TYPE UDT 1000
TITLE =PLC ==> 611U Process Data (POS Mode Control)
VERSION : 0.1


  STRUCT
   STW1 : STRUCT
    Bit_8 : BOOL ;	//Jog 1 On/Off
    Bit_9 : BOOL ;	//Jog 2 On/Off
    Bit_10 : BOOL ;	//Control Requested / No Control Requested
    Bit_11 : BOOL ;	//Start Referencing / Stop Referencing
    Bit_12 : BOOL ;	//Reserved
    Bit_13 : BOOL ;	//External Block Change
    Bit_14 : BOOL ;	//Reserved
    Bit_15 : BOOL ;	//Reserved
    Bit_0 : BOOL ;	//Enable / Off 1
    Bit_1 : BOOL ;	//Enable / Off 2
    Bit_2 : BOOL ;	//Enable / Off 3
    Bit_3 : BOOL ;	//Enable Inverter / Pulse Inhibit
    Bit_4 : BOOL ;	//Enable / Reject travel task
    Bit_5 : BOOL ;	//Enable / Immediatly stop
    Bit_6 : BOOL ;	//Activate Travel Block ( Edge )
    Bit_7 : BOOL ;	//Reset the Fault memory
   END_STRUCT ;
   SatzAnw : STRUCT
    BLKSEL : INT ;	//Block Selection 0 ~ 63
   END_STRUCT ;
   PosStw : STRUCT
    Bit_8 : BOOL ;	//Reserved
    Bit_9 : BOOL ;	//Reserved
    Bit_10 : BOOL ;	//Reserved
    Bit_11 : BOOL ;	//Reserved
    Bit_12 : BOOL ;	//Reserved
    Bit_13 : BOOL ;	//Reserved
    Bit_14 : BOOL ;	//Reserved
    Bit_15 : BOOL ;	//Reserved
    Bit_0 : BOOL ;	//Tracking Operation
    Bit_1 : BOOL ;	//Set Reference Point
    Bit_2 : BOOL ;	//Reference Cams
    Bit_3 : BOOL ;	//Acknowledgement, Function Bit
    Bit_4 : BOOL ;	//Reserved
    Bit_5 : BOOL ;	//Reserved
    Bit_6 : BOOL ;	//Reserved
    Bit_7 : BOOL ;	//Reserved
   END_STRUCT ;
   STW2 : STRUCT
    Bit_8 : BOOL ;	//Suppress Fault 608
    Bit_9 : BOOL ;	//Motor Data Change Over 1st input
    Bit_10 : BOOL ;	//Motor Data Change Over 2nd input
    Bit_11 : BOOL ;	//Motor Changed Over
    Bit_12 : BOOL ;	//Sign of Life Bit 0
    Bit_13 : BOOL ;	//Sign of Life Bit 1
    Bit_14 : BOOL ;	//Sign of Life Bit 2
    Bit_15 : BOOL ;	//Sign of Life Bit 3
    Bit_0 : BOOL ;	//Parameter Set Changeover Bit 0
    Bit_1 : BOOL ;	//Parameter Set Changeover Bit 1
    Bit_2 : BOOL ;	//Parameter Set Changeover Bit 2
    Bit_3 : BOOL ;	//First Speed Setpoint Filter off
    Bit_4 : BOOL ;	//Ramp up Time Zero
    Bit_5 : BOOL ;	//Reserved
    Bit_6 : BOOL ;	//Integrator inhibit, Speed Controller
    Bit_7 : BOOL ;	//Selection, Parking Axis
   END_STRUCT ;
   Over : STRUCT
    Override : INT ;	//Override Defined using P0833=>16384(dec) = 1%, 1638.4 = 0.1%
   END_STRUCT ;
   Temp1 : INT ;
   Temp2 : INT ;
   Temp3 : INT ;
   Temp4 : INT ;
   Temp5 : INT ;
  END_STRUCT ;
END_TYPE

TYPE UDT 2000
TITLE =POS Mode Control
VERSION : 0.1


  STRUCT
   ZSW1 : STRUCT
    Bit_8 : BOOL ;	//No Following error / Following error
    Bit_9 : BOOL ;	//Control requested / No Control Possible
    Bit_10 : BOOL ;	//Reference Point Reached / Outside ref.position
    Bit_11 : BOOL ;	//Reference Point Set / Reference Point Not Set
    Bit_12 : BOOL ;	//Setpoint Acknowledge (Edge)
    Bir_13 : BOOL ;	//Drive Stationary / Drive Active
    Bit_14 : BOOL ;	//Reserved
    Bit_15 : BOOL ;	//Reserved
    Bit_0 : BOOL ;	//Ready to Switch-on / Not ready to Switch-on
    Bit_1 : BOOL ;	//Ready or no Fault
    Bit_2 : BOOL ;	//Controller Enable Status
    Bit_3 : BOOL ;	//Fault Present / No Fault Present
    Bit_4 : BOOL ;	//No OFF2 Present / OFF2 Present
    Bit_5 : BOOL ;	//No OFF3 Present / OFF3 Present
    Bit_6 : BOOL ;	//Switch-on Inhibit / No Switch-on Inhibit
    Bit_7 : BOOL ;	//Alarm Present / No Alarm Present
   END_STRUCT ;
   AktSatz : STRUCT
    CURRBLK : INT ;	//Status Block Selection (0 ~ 63)
   END_STRUCT ;
   PosZsw : STRUCT
    Bit_8 : BOOL ;	//Cam Switching Signal 1
    Bit_9 : BOOL ;	//Cam Switching Signal 2
    Bit_10 : BOOL ;	//Direct Output 1 via the Traversing Block
    Bit_11 : BOOL ;	//Direct Output 2 via the Traversing Block
    Bit_12 : BOOL ;	//Reserved
    Bit_13 : BOOL ;	//Reserved
    Bit_14 : BOOL ;	//Reserved
    Bit_15 : BOOL ;	//Reserved
    Bit_0 : BOOL ;	//Tracking Mode Active
    Bit_1 : BOOL ;	//Velocity Limiting
    Bit_2 : BOOL ;	//Setpoint stationary
    Bit_3 : BOOL ;	//Function Bit
    Bit_4 : BOOL ;	//Axis Moves Forwards
    Bit_5 : BOOL ;	//Axis Moves Backwards
    Bit_6 : BOOL ;	//Minus Software Limit Switch Actuated
    Bit_7 : BOOL ;	//Plus Software Limit Switch Actuated
   END_STRUCT ;
   ZSW2 : STRUCT
    Bit_8 : BOOL ;	//Supress Fault 608 Active
    Bit_9 : BOOL ;	//Actual Motor 1st Signal
    Bit_10 : BOOL ;	//Actual Motor 2nd Signal
    Bit_11 : BOOL ;	//Reserved
    Bit_12 : BOOL ;	//Slave Sign of Life Bit 0
    Bit_13 : BOOL ;	//Slave Sign of Life Bit 1
    Bit_14 : BOOL ;	//Slave Sign of Life Bit 2
    Bit_15 : BOOL ;	//Slave Sign of Life Bit 3
    Bit_0 : BOOL ;	//Parameter Set Bit 0
    Bit_1 : BOOL ;	//Parameter Set Bit 1
    Bit_2 : BOOL ;	//Parameter Set Bit 2
    Bit_3 : BOOL ;	//First Speed Setpoint Filter Inactive
    Bit_4 : BOOL ;	//Ramp-Function gen Inactive
    Bit_5 : BOOL ;	//Open Holding Brake
    Bit_6 : BOOL ;	//Integrator Inhibit, Speed Controller
    Bit_7 : BOOL ;	//Parking Axis Selected
   END_STRUCT ;
   MessW : STRUCT
    Bit_8 : BOOL ;	//|nset| = |nact |
    Bit_9 : BOOL ;	//Reserved
    Bit_10 : BOOL ;	//Power Module Current Not Limited
    Bit_11 : BOOL ;	//Reserved
    Bit_12 : BOOL ;	//Reserved
    Bit_13 : BOOL ;	//Pulse Enabled
    Bit_14 : BOOL ;	//Reserved
    Bit_15 : BOOL ;	//Reserved
    Bit_0 : BOOL ;	//Ramp-up Completed
    Bit_1 : BOOL ;	//|M| < Mx
    Bit_2 : BOOL ;	//|nact| < nmin
    Bit_3 : BOOL ;	//|nact| < nx
    Bit_4 : BOOL ;	//DC Link Monitoring VDC link > Vx
    Bit_5 : BOOL ;	//Variable Message Function
    Bit_6 : BOOL ;	//Motor Overtemperature Pre-Alarm
    Bit_7 : BOOL ;	//Heatsink Temperature Pre-Alarm
   END_STRUCT ;
   XactP1 : WORD ;	//Position Actual Value (Pos Mode) Word1
   XactP2 : WORD ;	//Position Actual Value (Pos Mode) Word2
   Temp1 : INT ;
   Temp2 : INT ;
   Temp3 : INT ;
  END_STRUCT ;
END_TYPE

DATA_BLOCK DB 2
TITLE =
VERSION : 0.1


  STRUCT
   SEND1_DATA : STRUCT 	//Temporary placeholder variable
    SEND_DONE : BOOL ;
    SEND_ERROR : BOOL ;
    SEND_SCAN : BOOL ;
    SEND_ACT : BOOL ;
    SEND_SP1 : BOOL ;
    SEND_SP2 : BOOL ;
    SEND_SP3 : BOOL ;
    SEND_SP4 : BOOL ;
    SEND_STATUS : WORD ;
    SPARE2 : ARRAY  [0 .. 2 ] OF WORD ;
   END_STRUCT ;
   SEND2_DATA : STRUCT 	//Temporary placeholder variable
    SEND_DONE : BOOL ;
    SEND_ERROR : BOOL ;
    SEND_SCAN : BOOL ;
    SEND_ACT : BOOL ;
    SEND_SP1 : BOOL ;
    SEND_SP2 : BOOL ;
    SEND_SP3 : BOOL ;
    SEND_SP4 : BOOL ;
    SEND_STATUS : WORD ;
    SPARE2 : ARRAY  [0 .. 2 ] OF WORD ;
   END_STRUCT ;
   SEND3_DATA : STRUCT 	//Temporary placeholder variable
    SEND_DONE : BOOL ;
    SEND_ERROR : BOOL ;
    SEND_SCAN : BOOL ;
    SEND_ACT : BOOL ;
    SEND_SP1 : BOOL ;
    SEND_SP2 : BOOL ;
    SEND_SP3 : BOOL ;
    SEND_SP4 : BOOL ;
    SEND_STATUS : WORD ;
    SPARE2 : ARRAY  [0 .. 2 ] OF WORD ;
   END_STRUCT ;
   SEND4_DATA : STRUCT 	//Temporary placeholder variable
    SEND_DONE : BOOL ;
    SEND_ERROR : BOOL ;
    SEND_SCAN : BOOL ;
    SEND_ACT : BOOL ;
    SEND_SP1 : BOOL ;
    SEND_SP2 : BOOL ;
    SEND_SP3 : BOOL ;
    SEND_SP4 : BOOL ;
    SEND_STATUS : WORD ;
    SPARE2 : ARRAY  [0 .. 2 ] OF WORD ;
   END_STRUCT ;
   SEND5_DATA : STRUCT 	//Temporary placeholder variable
    SEND_DONE : BOOL ;
    SEND_ERROR : BOOL ;
    SEND_SCAN : BOOL ;
    SEND_ACT : BOOL ;
    SEND_SP1 : BOOL ;
    SEND_SP2 : BOOL ;
    SEND_SP3 : BOOL ;
    SEND_SP4 : BOOL ;
    SEND_STATUS : WORD ;
    SPARE2 : ARRAY  [0 .. 2 ] OF WORD ;
   END_STRUCT ;
   SEND6_DATA : STRUCT 	//Temporary placeholder variable
    SEND_DONE : BOOL ;
    SEND_ERROR : BOOL ;
    SEND_SCAN : BOOL ;
    SEND_ACT : BOOL ;
    SEND_SP1 : BOOL ;
    SEND_SP2 : BOOL ;
    SEND_SP3 : BOOL ;
    SEND_SP4 : BOOL ;
    SEND_STATUS : WORD ;
    SPARE2 : ARRAY  [0 .. 2 ] OF WORD ;
   END_STRUCT ;
   SEND7_DATA : STRUCT 	//Temporary placeholder variable
    SEND_DONE : BOOL ;
    SEND_ERROR : BOOL ;
    SEND_SCAN : BOOL ;
    SEND_ACT : BOOL ;
    SEND_SP1 : BOOL ;
    SEND_SP2 : BOOL ;
    SEND_SP3 : BOOL ;
    SEND_SP4 : BOOL ;
    SEND_STATUS : WORD ;
    SPARE2 : ARRAY  [0 .. 2 ] OF WORD ;
   END_STRUCT ;
   SEND8_DATA : STRUCT 	//Temporary placeholder variable
    SEND_DONE : BOOL ;
    SEND_ERROR : BOOL ;
    SEND_SCAN : BOOL ;
    SEND_ACT : BOOL ;
    SEND_SP1 : BOOL ;
    SEND_SP2 : BOOL ;
    SEND_SP3 : BOOL ;
    SEND_SP4 : BOOL ;
    SEND_STATUS : WORD ;
    SPARE2 : ARRAY  [0 .. 2 ] OF WORD ;
   END_STRUCT ;
   SEND9_DATA : STRUCT 	//Temporary placeholder variable
    SEND_DONE : BOOL ;
    SEND_ERROR : BOOL ;
    SEND_SCAN : BOOL ;
    SEND_ACT : BOOL ;
    SEND_SP1 : BOOL ;
    SEND_SP2 : BOOL ;
    SEND_SP3 : BOOL ;
    SEND_SP4 : BOOL ;
    SEND_STATUS : WORD ;
    SPARE2 : ARRAY  [0 .. 2 ] OF WORD ;
   END_STRUCT ;
   SEND10_DATA : STRUCT 	//Temporary placeholder variable
    SEND_DONE : BOOL ;
    SEND_ERROR : BOOL ;
    SEND_SCAN : BOOL ;
    SEND_ACT : BOOL ;
    SEND_SP1 : BOOL ;
    SEND_SP2 : BOOL ;
    SEND_SP3 : BOOL ;
    SEND_SP4 : BOOL ;
    SEND_STATUS : WORD ;
    SPARE2 : ARRAY  [0 .. 2 ] OF WORD ;
   END_STRUCT ;
   RECV1_DATA : STRUCT 	//Temporary placeholder variable
    RECV_NDR : BOOL ;
    RECV_ERROR : BOOL ;
    RECV_DATA3 : BOOL ;
    RECV_DATA4 : BOOL ;
    RECV_DATA5 : BOOL ;
    RECV_DATA6 : BOOL ;
    RECV_DATA7 : BOOL ;
    RECV_DATA8 : BOOL ;
    RECV_STATUS : WORD ;
    RECV_LEN : INT ;
    SPARE2 : ARRAY  [0 .. 3 ] OF BYTE ;
   END_STRUCT ;
   RECV2_DATA : STRUCT 	//Temporary placeholder variable
    RECV_NDR : BOOL ;
    RECV_ERROR : BOOL ;
    RECV_DATA3 : BOOL ;
    RECV_DATA4 : BOOL ;
    RECV_DATA5 : BOOL ;
    RECV_DATA6 : BOOL ;
    RECV_DATA7 : BOOL ;
    RECV_DATA8 : BOOL ;
    RECV_STATUS : WORD ;
    RECV_LEN : INT ;
    SPARE2 : ARRAY  [0 .. 3 ] OF BYTE ;
   END_STRUCT ;
   RECV3_DATA : STRUCT 	//Temporary placeholder variable
    RECV_NDR : BOOL ;
    RECV_ERROR : BOOL ;
    RECV_DATA3 : BOOL ;
    RECV_DATA4 : BOOL ;
    RECV_DATA5 : BOOL ;
    RECV_DATA6 : BOOL ;
    RECV_DATA7 : BOOL ;
    RECV_DATA8 : BOOL ;
    RECV_STATUS : WORD ;
    RECV_LEN : INT ;
    SPARE2 : ARRAY  [0 .. 3 ] OF BYTE ;
   END_STRUCT ;
   RECV4_DATA : STRUCT 	//Temporary placeholder variable
    RECV_NDR : BOOL ;
    RECV_ERROR : BOOL ;
    RECV_DATA3 : BOOL ;
    RECV_DATA4 : BOOL ;
    RECV_DATA5 : BOOL ;
    RECV_DATA6 : BOOL ;
    RECV_DATA7 : BOOL ;
    RECV_DATA8 : BOOL ;
    RECV_STATUS : WORD ;
    RECV_LEN : INT ;
    SPARE2 : ARRAY  [0 .. 3 ] OF BYTE ;
   END_STRUCT ;
   RECV5_DATA : STRUCT 	//Temporary placeholder variable
    RECV_NDR : BOOL ;
    RECV_ERROR : BOOL ;
    RECV_DATA3 : BOOL ;
    RECV_DATA4 : BOOL ;
    RECV_DATA5 : BOOL ;
    RECV_DATA6 : BOOL ;
    RECV_DATA7 : BOOL ;
    RECV_DATA8 : BOOL ;
    RECV_STATUS : WORD ;
    RECV_LEN : INT ;
    SPARE2 : ARRAY  [0 .. 3 ] OF BYTE ;
   END_STRUCT ;
   RECV6_DATA : STRUCT 	//Temporary placeholder variable
    RECV_NDR : BOOL ;
    RECV_ERROR : BOOL ;
    RECV_DATA3 : BOOL ;
    RECV_DATA4 : BOOL ;
    RECV_DATA5 : BOOL ;
    RECV_DATA6 : BOOL ;
    RECV_DATA7 : BOOL ;
    RECV_DATA8 : BOOL ;
    RECV_STATUS : WORD ;
    RECV_LEN : INT ;
    SPARE2 : ARRAY  [0 .. 3 ] OF BYTE ;
   END_STRUCT ;
   RECV7_DATA : STRUCT 	//Temporary placeholder variable
    RECV_NDR : BOOL ;
    RECV_ERROR : BOOL ;
    RECV_DATA3 : BOOL ;
    RECV_DATA4 : BOOL ;
    RECV_DATA5 : BOOL ;
    RECV_DATA6 : BOOL ;
    RECV_DATA7 : BOOL ;
    RECV_DATA8 : BOOL ;
    RECV_STATUS : WORD ;
    RECV_LEN : INT ;
    SPARE2 : ARRAY  [0 .. 3 ] OF BYTE ;
   END_STRUCT ;
   RECV8_DATA : STRUCT 	//Temporary placeholder variable
    RECV_NDR : BOOL ;
    RECV_ERROR : BOOL ;
    RECV_DATA3 : BOOL ;
    RECV_DATA4 : BOOL ;
    RECV_DATA5 : BOOL ;
    RECV_DATA6 : BOOL ;
    RECV_DATA7 : BOOL ;
    RECV_DATA8 : BOOL ;
    RECV_STATUS : WORD ;
    RECV_LEN : INT ;
    SPARE2 : ARRAY  [0 .. 3 ] OF BYTE ;
   END_STRUCT ;
   RECV9_DATA : STRUCT 	//Temporary placeholder variable
    RECV_NDR : BOOL ;
    RECV_ERROR : BOOL ;
    RECV_DATA3 : BOOL ;
    RECV_DATA4 : BOOL ;
    RECV_DATA5 : BOOL ;
    RECV_DATA6 : BOOL ;
    RECV_DATA7 : BOOL ;
    RECV_DATA8 : BOOL ;
    RECV_STATUS : WORD ;
    RECV_LEN : INT ;
    SPARE2 : ARRAY  [0 .. 3 ] OF BYTE ;
   END_STRUCT ;
   RECV10_DATA : STRUCT 	//Temporary placeholder variable
    RECV_NDR : BOOL ;
    RECV_ERROR : BOOL ;
    RECV_DATA3 : BOOL ;
    RECV_DATA4 : BOOL ;
    RECV_DATA5 : BOOL ;
    RECV_DATA6 : BOOL ;
    RECV_DATA7 : BOOL ;
    RECV_DATA8 : BOOL ;
    RECV_STATUS : WORD ;
    RECV_LEN : INT ;
    SPARE2 : ARRAY  [0 .. 3 ] OF BYTE ;
   END_STRUCT ;
   SEND11_DATA : STRUCT 	//Temporary placeholder variable
    SEND_DONE : BOOL ;
    SEND_ERROR : BOOL ;
    SEND_SCAN : BOOL ;
    SEND_ACT : BOOL ;
    SEND_SP1 : BOOL ;
    SEND_SP2 : BOOL ;
    SEND_SP3 : BOOL ;
    SEND_SP4 : BOOL ;
    SEND_STATUS : WORD ;
    SPARE2 : ARRAY  [0 .. 2 ] OF WORD ;
   END_STRUCT ;
   SEND12_DATA : STRUCT 	//Temporary placeholder variable
    SEND_DONE : BOOL ;
    SEND_ERROR : BOOL ;
    SEND_SCAN : BOOL ;
    SEND_ACT : BOOL ;
    SEND_SP1 : BOOL ;
    SEND_SP2 : BOOL ;
    SEND_SP3 : BOOL ;
    SEND_SP4 : BOOL ;
    SEND_STATUS : WORD ;
    SPARE2 : ARRAY  [0 .. 2 ] OF WORD ;
   END_STRUCT ;
   SEND13_DATA : STRUCT 	//Temporary placeholder variable
    SEND_DONE : BOOL ;
    SEND_ERROR : BOOL ;
    SEND_SCAN : BOOL ;
    SEND_ACT : BOOL ;
    SEND_SP1 : BOOL ;
    SEND_SP2 : BOOL ;
    SEND_SP3 : BOOL ;
    SEND_SP4 : BOOL ;
    SEND_STATUS : WORD ;
    SPARE2 : ARRAY  [0 .. 2 ] OF WORD ;
   END_STRUCT ;
   SEND14_DATA : STRUCT 	//Temporary placeholder variable
    SEND_DONE : BOOL ;
    SEND_ERROR : BOOL ;
    SEND_SCAN : BOOL ;
    SEND_ACT : BOOL ;
    SEND_SP1 : BOOL ;
    SEND_SP2 : BOOL ;
    SEND_SP3 : BOOL ;
    SEND_SP4 : BOOL ;
    SEND_STATUS : WORD ;
    SPARE2 : ARRAY  [0 .. 2 ] OF WORD ;
   END_STRUCT ;
   SEND15_DATA : STRUCT 	//Temporary placeholder variable
    SEND_DONE : BOOL ;
    SEND_ERROR : BOOL ;
    SEND_SCAN : BOOL ;
    SEND_ACT : BOOL ;
    SEND_SP1 : BOOL ;
    SEND_SP2 : BOOL ;
    SEND_SP3 : BOOL ;
    SEND_SP4 : BOOL ;
    SEND_STATUS : WORD ;
    SPARE2 : ARRAY  [0 .. 2 ] OF WORD ;
   END_STRUCT ;
   SEND16_DATA : STRUCT 	//Temporary placeholder variable
    SEND_DONE : BOOL ;
    SEND_ERROR : BOOL ;
    SEND_SCAN : BOOL ;
    SEND_ACT : BOOL ;
    SEND_SP1 : BOOL ;
    SEND_SP2 : BOOL ;
    SEND_SP3 : BOOL ;
    SEND_SP4 : BOOL ;
    SEND_STATUS : WORD ;
    SPARE2 : ARRAY  [0 .. 2 ] OF WORD ;
   END_STRUCT ;
   SEND17_DATA : STRUCT 	//Temporary placeholder variable
    SEND_DONE : BOOL ;
    SEND_ERROR : BOOL ;
    SEND_SCAN : BOOL ;
    SEND_ACT : BOOL ;
    SEND_SP1 : BOOL ;
    SEND_SP2 : BOOL ;
    SEND_SP3 : BOOL ;
    SEND_SP4 : BOOL ;
    SEND_STATUS : WORD ;
    SPARE2 : ARRAY  [0 .. 2 ] OF WORD ;
   END_STRUCT ;
   SEND18_DATA : STRUCT 	//Temporary placeholder variable
    SEND_DONE : BOOL ;
    SEND_ERROR : BOOL ;
    SEND_SCAN : BOOL ;
    SEND_ACT : BOOL ;
    SEND_SP1 : BOOL ;
    SEND_SP2 : BOOL ;
    SEND_SP3 : BOOL ;
    SEND_SP4 : BOOL ;
    SEND_STATUS : WORD ;
    SPARE2 : ARRAY  [0 .. 2 ] OF WORD ;
   END_STRUCT ;
   SEND19_DATA : STRUCT 	//Temporary placeholder variable
    SEND_DONE : BOOL ;
    SEND_ERROR : BOOL ;
    SEND_SCAN : BOOL ;
    SEND_ACT : BOOL ;
    SEND_SP1 : BOOL ;
    SEND_SP2 : BOOL ;
    SEND_SP3 : BOOL ;
    SEND_SP4 : BOOL ;
    SEND_STATUS : WORD ;
    SPARE2 : ARRAY  [0 .. 2 ] OF WORD ;
   END_STRUCT ;
   SEND20_DATA : STRUCT 	//Temporary placeholder variable
    SEND_DONE : BOOL ;
    SEND_ERROR : BOOL ;
    SEND_SCAN : BOOL ;
    SEND_ACT : BOOL ;
    SEND_SP1 : BOOL ;
    SEND_SP2 : BOOL ;
    SEND_SP3 : BOOL ;
    SEND_SP4 : BOOL ;
    SEND_STATUS : WORD ;
    SPARE2 : ARRAY  [0 .. 2 ] OF WORD ;
   END_STRUCT ;
   RECV11_DATA : STRUCT 	//Temporary placeholder variable
    RECV_NDR : BOOL ;
    RECV_ERROR : BOOL ;
    RECV_DATA3 : BOOL ;
    RECV_DATA4 : BOOL ;
    RECV_DATA5 : BOOL ;
    RECV_DATA6 : BOOL ;
    RECV_DATA7 : BOOL ;
    RECV_DATA8 : BOOL ;
    RECV_STATUS : WORD ;
    RECV_LEN : INT ;
    SPARE2 : ARRAY  [0 .. 3 ] OF BYTE ;
   END_STRUCT ;
   RECV12_DATA : STRUCT 	//Temporary placeholder variable
    RECV_NDR : BOOL ;
    RECV_ERROR : BOOL ;
    RECV_DATA3 : BOOL ;
    RECV_DATA4 : BOOL ;
    RECV_DATA5 : BOOL ;
    RECV_DATA6 : BOOL ;
    RECV_DATA7 : BOOL ;
    RECV_DATA8 : BOOL ;
    RECV_STATUS : WORD ;
    RECV_LEN : INT ;
    SPARE2 : ARRAY  [0 .. 3 ] OF BYTE ;
   END_STRUCT ;
   RECV13_DATA : STRUCT 	//Temporary placeholder variable
    RECV_NDR : BOOL ;
    RECV_ERROR : BOOL ;
    RECV_DATA3 : BOOL ;
    RECV_DATA4 : BOOL ;
    RECV_DATA5 : BOOL ;
    RECV_DATA6 : BOOL ;
    RECV_DATA7 : BOOL ;
    RECV_DATA8 : BOOL ;
    RECV_STATUS : WORD ;
    RECV_LEN : INT ;
    SPARE2 : ARRAY  [0 .. 3 ] OF BYTE ;
   END_STRUCT ;
   RECV14_DATA : STRUCT 	//Temporary placeholder variable
    RECV_NDR : BOOL ;
    RECV_ERROR : BOOL ;
    RECV_DATA3 : BOOL ;
    RECV_DATA4 : BOOL ;
    RECV_DATA5 : BOOL ;
    RECV_DATA6 : BOOL ;
    RECV_DATA7 : BOOL ;
    RECV_DATA8 : BOOL ;
    RECV_STATUS : WORD ;
    RECV_LEN : INT ;
    SPARE2 : ARRAY  [0 .. 3 ] OF BYTE ;
   END_STRUCT ;
   RECV15_DATA : STRUCT 	//Temporary placeholder variable
    RECV_NDR : BOOL ;
    RECV_ERROR : BOOL ;
    RECV_DATA3 : BOOL ;
    RECV_DATA4 : BOOL ;
    RECV_DATA5 : BOOL ;
    RECV_DATA6 : BOOL ;
    RECV_DATA7 : BOOL ;
    RECV_DATA8 : BOOL ;
    RECV_STATUS : WORD ;
    RECV_LEN : INT ;
    SPARE2 : ARRAY  [0 .. 3 ] OF BYTE ;
   END_STRUCT ;
   RECV16_DATA : STRUCT 	//Temporary placeholder variable
    RECV_NDR : BOOL ;
    RECV_ERROR : BOOL ;
    RECV_DATA3 : BOOL ;
    RECV_DATA4 : BOOL ;
    RECV_DATA5 : BOOL ;
    RECV_DATA6 : BOOL ;
    RECV_DATA7 : BOOL ;
    RECV_DATA8 : BOOL ;
    RECV_STATUS : WORD ;
    RECV_LEN : INT ;
    SPARE2 : ARRAY  [0 .. 3 ] OF BYTE ;
   END_STRUCT ;
   RECV17_DATA : STRUCT 	//Temporary placeholder variable
    RECV_NDR : BOOL ;
    RECV_ERROR : BOOL ;
    RECV_DATA3 : BOOL ;
    RECV_DATA4 : BOOL ;
    RECV_DATA5 : BOOL ;
    RECV_DATA6 : BOOL ;
    RECV_DATA7 : BOOL ;
    RECV_DATA8 : BOOL ;
    RECV_STATUS : WORD ;
    RECV_LEN : INT ;
    SPARE2 : ARRAY  [0 .. 3 ] OF BYTE ;
   END_STRUCT ;
   RECV18_DATA : STRUCT 	//Temporary placeholder variable
    RECV_NDR : BOOL ;
    RECV_ERROR : BOOL ;
    RECV_DATA3 : BOOL ;
    RECV_DATA4 : BOOL ;
    RECV_DATA5 : BOOL ;
    RECV_DATA6 : BOOL ;
    RECV_DATA7 : BOOL ;
    RECV_DATA8 : BOOL ;
    RECV_STATUS : WORD ;
    RECV_LEN : INT ;
    SPARE2 : ARRAY  [0 .. 3 ] OF BYTE ;
   END_STRUCT ;
   RECV19_DATA : STRUCT 	//Temporary placeholder variable
    RECV_NDR : BOOL ;
    RECV_ERROR : BOOL ;
    RECV_DATA3 : BOOL ;
    RECV_DATA4 : BOOL ;
    RECV_DATA5 : BOOL ;
    RECV_DATA6 : BOOL ;
    RECV_DATA7 : BOOL ;
    RECV_DATA8 : BOOL ;
    RECV_STATUS : WORD ;
    RECV_LEN : INT ;
    SPARE2 : ARRAY  [0 .. 3 ] OF BYTE ;
   END_STRUCT ;
   RECV20_DATA : STRUCT 	//Temporary placeholder variable
    RECV_NDR : BOOL ;
    RECV_ERROR : BOOL ;
    RECV_DATA3 : BOOL ;
    RECV_DATA4 : BOOL ;
    RECV_DATA5 : BOOL ;
    RECV_DATA6 : BOOL ;
    RECV_DATA7 : BOOL ;
    RECV_DATA8 : BOOL ;
    RECV_STATUS : WORD ;
    RECV_LEN : INT ;
    SPARE2 : ARRAY  [0 .. 3 ] OF BYTE ;
   END_STRUCT ;
  END_STRUCT ;
BEGIN
   SEND1_DATA.SEND_DONE := FALSE;
   SEND1_DATA.SEND_ERROR := FALSE;
   SEND1_DATA.SEND_SCAN := FALSE;
   SEND1_DATA.SEND_ACT := FALSE;
   SEND1_DATA.SEND_SP1 := FALSE;
   SEND1_DATA.SEND_SP2 := FALSE;
   SEND1_DATA.SEND_SP3 := FALSE;
   SEND1_DATA.SEND_SP4 := FALSE;
   SEND1_DATA.SEND_STATUS := W#16#0;
   SEND1_DATA.SPARE2[0] := W#16#0;
   SEND1_DATA.SPARE2[1] := W#16#0;
   SEND1_DATA.SPARE2[2] := W#16#0;
   SEND2_DATA.SEND_DONE := FALSE;
   SEND2_DATA.SEND_ERROR := FALSE;
   SEND2_DATA.SEND_SCAN := FALSE;
   SEND2_DATA.SEND_ACT := FALSE;
   SEND2_DATA.SEND_SP1 := FALSE;
   SEND2_DATA.SEND_SP2 := FALSE;
   SEND2_DATA.SEND_SP3 := FALSE;
   SEND2_DATA.SEND_SP4 := FALSE;
   SEND2_DATA.SEND_STATUS := W#16#0;
   SEND2_DATA.SPARE2[0] := W#16#0;
   SEND2_DATA.SPARE2[1] := W#16#0;
   SEND2_DATA.SPARE2[2] := W#16#0;
   SEND3_DATA.SEND_DONE := FALSE;
   SEND3_DATA.SEND_ERROR := FALSE;
   SEND3_DATA.SEND_SCAN := FALSE;
   SEND3_DATA.SEND_ACT := FALSE;
   SEND3_DATA.SEND_SP1 := FALSE;
   SEND3_DATA.SEND_SP2 := FALSE;
   SEND3_DATA.SEND_SP3 := FALSE;
   SEND3_DATA.SEND_SP4 := FALSE;
   SEND3_DATA.SEND_STATUS := W#16#0;
   SEND3_DATA.SPARE2[0] := W#16#0;
   SEND3_DATA.SPARE2[1] := W#16#0;
   SEND3_DATA.SPARE2[2] := W#16#0;
   SEND4_DATA.SEND_DONE := FALSE;
   SEND4_DATA.SEND_ERROR := FALSE;
   SEND4_DATA.SEND_SCAN := FALSE;
   SEND4_DATA.SEND_ACT := FALSE;
   SEND4_DATA.SEND_SP1 := FALSE;
   SEND4_DATA.SEND_SP2 := FALSE;
   SEND4_DATA.SEND_SP3 := FALSE;
   SEND4_DATA.SEND_SP4 := FALSE;
   SEND4_DATA.SEND_STATUS := W#16#0;
   SEND4_DATA.SPARE2[0] := W#16#0;
   SEND4_DATA.SPARE2[1] := W#16#0;
   SEND4_DATA.SPARE2[2] := W#16#0;
   SEND5_DATA.SEND_DONE := FALSE;
   SEND5_DATA.SEND_ERROR := FALSE;
   SEND5_DATA.SEND_SCAN := FALSE;
   SEND5_DATA.SEND_ACT := FALSE;
   SEND5_DATA.SEND_SP1 := FALSE;
   SEND5_DATA.SEND_SP2 := FALSE;
   SEND5_DATA.SEND_SP3 := FALSE;
   SEND5_DATA.SEND_SP4 := FALSE;
   SEND5_DATA.SEND_STATUS := W#16#0;
   SEND5_DATA.SPARE2[0] := W#16#0;
   SEND5_DATA.SPARE2[1] := W#16#0;
   SEND5_DATA.SPARE2[2] := W#16#0;
   SEND6_DATA.SEND_DONE := FALSE;
   SEND6_DATA.SEND_ERROR := FALSE;
   SEND6_DATA.SEND_SCAN := FALSE;
   SEND6_DATA.SEND_ACT := FALSE;
   SEND6_DATA.SEND_SP1 := FALSE;
   SEND6_DATA.SEND_SP2 := FALSE;
   SEND6_DATA.SEND_SP3 := FALSE;
   SEND6_DATA.SEND_SP4 := FALSE;
   SEND6_DATA.SEND_STATUS := W#16#0;
   SEND6_DATA.SPARE2[0] := W#16#0;
   SEND6_DATA.SPARE2[1] := W#16#0;
   SEND6_DATA.SPARE2[2] := W#16#0;
   SEND7_DATA.SEND_DONE := FALSE;
   SEND7_DATA.SEND_ERROR := FALSE;
   SEND7_DATA.SEND_SCAN := FALSE;
   SEND7_DATA.SEND_ACT := FALSE;
   SEND7_DATA.SEND_SP1 := FALSE;
   SEND7_DATA.SEND_SP2 := FALSE;
   SEND7_DATA.SEND_SP3 := FALSE;
   SEND7_DATA.SEND_SP4 := FALSE;
   SEND7_DATA.SEND_STATUS := W#16#0;
   SEND7_DATA.SPARE2[0] := W#16#0;
   SEND7_DATA.SPARE2[1] := W#16#0;
   SEND7_DATA.SPARE2[2] := W#16#0;
   SEND8_DATA.SEND_DONE := FALSE;
   SEND8_DATA.SEND_ERROR := FALSE;
   SEND8_DATA.SEND_SCAN := FALSE;
   SEND8_DATA.SEND_ACT := FALSE;
   SEND8_DATA.SEND_SP1 := FALSE;
   SEND8_DATA.SEND_SP2 := FALSE;
   SEND8_DATA.SEND_SP3 := FALSE;
   SEND8_DATA.SEND_SP4 := FALSE;
   SEND8_DATA.SEND_STATUS := W#16#0;
   SEND8_DATA.SPARE2[0] := W#16#0;
   SEND8_DATA.SPARE2[1] := W#16#0;
   SEND8_DATA.SPARE2[2] := W#16#0;
   SEND9_DATA.SEND_DONE := FALSE;
   SEND9_DATA.SEND_ERROR := FALSE;
   SEND9_DATA.SEND_SCAN := FALSE;
   SEND9_DATA.SEND_ACT := FALSE;
   SEND9_DATA.SEND_SP1 := FALSE;
   SEND9_DATA.SEND_SP2 := FALSE;
   SEND9_DATA.SEND_SP3 := FALSE;
   SEND9_DATA.SEND_SP4 := FALSE;
   SEND9_DATA.SEND_STATUS := W#16#0;
   SEND9_DATA.SPARE2[0] := W#16#0;
   SEND9_DATA.SPARE2[1] := W#16#0;
   SEND9_DATA.SPARE2[2] := W#16#0;
   SEND10_DATA.SEND_DONE := FALSE;
   SEND10_DATA.SEND_ERROR := FALSE;
   SEND10_DATA.SEND_SCAN := FALSE;
   SEND10_DATA.SEND_ACT := FALSE;
   SEND10_DATA.SEND_SP1 := FALSE;
   SEND10_DATA.SEND_SP2 := FALSE;
   SEND10_DATA.SEND_SP3 := FALSE;
   SEND10_DATA.SEND_SP4 := FALSE;
   SEND10_DATA.SEND_STATUS := W#16#0;
   SEND10_DATA.SPARE2[0] := W#16#0;
   SEND10_DATA.SPARE2[1] := W#16#0;
   SEND10_DATA.SPARE2[2] := W#16#0;
   RECV1_DATA.RECV_NDR := FALSE;
   RECV1_DATA.RECV_ERROR := FALSE;
   RECV1_DATA.RECV_DATA3 := FALSE;
   RECV1_DATA.RECV_DATA4 := FALSE;
   RECV1_DATA.RECV_DATA5 := FALSE;
   RECV1_DATA.RECV_DATA6 := FALSE;
   RECV1_DATA.RECV_DATA7 := FALSE;
   RECV1_DATA.RECV_DATA8 := FALSE;
   RECV1_DATA.RECV_STATUS := W#16#0;
   RECV1_DATA.RECV_LEN := 0;
   RECV1_DATA.SPARE2[0] := B#16#0;
   RECV1_DATA.SPARE2[1] := B#16#0;
   RECV1_DATA.SPARE2[2] := B#16#0;
   RECV1_DATA.SPARE2[3] := B#16#0;
   RECV2_DATA.RECV_NDR := FALSE;
   RECV2_DATA.RECV_ERROR := FALSE;
   RECV2_DATA.RECV_DATA3 := FALSE;
   RECV2_DATA.RECV_DATA4 := FALSE;
   RECV2_DATA.RECV_DATA5 := FALSE;
   RECV2_DATA.RECV_DATA6 := FALSE;
   RECV2_DATA.RECV_DATA7 := FALSE;
   RECV2_DATA.RECV_DATA8 := FALSE;
   RECV2_DATA.RECV_STATUS := W#16#0;
   RECV2_DATA.RECV_LEN := 0;
   RECV2_DATA.SPARE2[0] := B#16#0;
   RECV2_DATA.SPARE2[1] := B#16#0;
   RECV2_DATA.SPARE2[2] := B#16#0;
   RECV2_DATA.SPARE2[3] := B#16#0;
   RECV3_DATA.RECV_NDR := FALSE;
   RECV3_DATA.RECV_ERROR := FALSE;
   RECV3_DATA.RECV_DATA3 := FALSE;
   RECV3_DATA.RECV_DATA4 := FALSE;
   RECV3_DATA.RECV_DATA5 := FALSE;
   RECV3_DATA.RECV_DATA6 := FALSE;
   RECV3_DATA.RECV_DATA7 := FALSE;
   RECV3_DATA.RECV_DATA8 := FALSE;
   RECV3_DATA.RECV_STATUS := W#16#0;
   RECV3_DATA.RECV_LEN := 0;
   RECV3_DATA.SPARE2[0] := B#16#0;
   RECV3_DATA.SPARE2[1] := B#16#0;
   RECV3_DATA.SPARE2[2] := B#16#0;
   RECV3_DATA.SPARE2[3] := B#16#0;
   RECV4_DATA.RECV_NDR := FALSE;
   RECV4_DATA.RECV_ERROR := FALSE;
   RECV4_DATA.RECV_DATA3 := FALSE;
   RECV4_DATA.RECV_DATA4 := FALSE;
   RECV4_DATA.RECV_DATA5 := FALSE;
   RECV4_DATA.RECV_DATA6 := FALSE;
   RECV4_DATA.RECV_DATA7 := FALSE;
   RECV4_DATA.RECV_DATA8 := FALSE;
   RECV4_DATA.RECV_STATUS := W#16#0;
   RECV4_DATA.RECV_LEN := 0;
   RECV4_DATA.SPARE2[0] := B#16#0;
   RECV4_DATA.SPARE2[1] := B#16#0;
   RECV4_DATA.SPARE2[2] := B#16#0;
   RECV4_DATA.SPARE2[3] := B#16#0;
   RECV5_DATA.RECV_NDR := FALSE;
   RECV5_DATA.RECV_ERROR := FALSE;
   RECV5_DATA.RECV_DATA3 := FALSE;
   RECV5_DATA.RECV_DATA4 := FALSE;
   RECV5_DATA.RECV_DATA5 := FALSE;
   RECV5_DATA.RECV_DATA6 := FALSE;
   RECV5_DATA.RECV_DATA7 := FALSE;
   RECV5_DATA.RECV_DATA8 := FALSE;
   RECV5_DATA.RECV_STATUS := W#16#0;
   RECV5_DATA.RECV_LEN := 0;
   RECV5_DATA.SPARE2[0] := B#16#0;
   RECV5_DATA.SPARE2[1] := B#16#0;
   RECV5_DATA.SPARE2[2] := B#16#0;
   RECV5_DATA.SPARE2[3] := B#16#0;
   RECV6_DATA.RECV_NDR := FALSE;
   RECV6_DATA.RECV_ERROR := FALSE;
   RECV6_DATA.RECV_DATA3 := FALSE;
   RECV6_DATA.RECV_DATA4 := FALSE;
   RECV6_DATA.RECV_DATA5 := FALSE;
   RECV6_DATA.RECV_DATA6 := FALSE;
   RECV6_DATA.RECV_DATA7 := FALSE;
   RECV6_DATA.RECV_DATA8 := FALSE;
   RECV6_DATA.RECV_STATUS := W#16#0;
   RECV6_DATA.RECV_LEN := 0;
   RECV6_DATA.SPARE2[0] := B#16#0;
   RECV6_DATA.SPARE2[1] := B#16#0;
   RECV6_DATA.SPARE2[2] := B#16#0;
   RECV6_DATA.SPARE2[3] := B#16#0;
   RECV7_DATA.RECV_NDR := FALSE;
   RECV7_DATA.RECV_ERROR := FALSE;
   RECV7_DATA.RECV_DATA3 := FALSE;
   RECV7_DATA.RECV_DATA4 := FALSE;
   RECV7_DATA.RECV_DATA5 := FALSE;
   RECV7_DATA.RECV_DATA6 := FALSE;
   RECV7_DATA.RECV_DATA7 := FALSE;
   RECV7_DATA.RECV_DATA8 := FALSE;
   RECV7_DATA.RECV_STATUS := W#16#0;
   RECV7_DATA.RECV_LEN := 0;
   RECV7_DATA.SPARE2[0] := B#16#0;
   RECV7_DATA.SPARE2[1] := B#16#0;
   RECV7_DATA.SPARE2[2] := B#16#0;
   RECV7_DATA.SPARE2[3] := B#16#0;
   RECV8_DATA.RECV_NDR := FALSE;
   RECV8_DATA.RECV_ERROR := FALSE;
   RECV8_DATA.RECV_DATA3 := FALSE;
   RECV8_DATA.RECV_DATA4 := FALSE;
   RECV8_DATA.RECV_DATA5 := FALSE;
   RECV8_DATA.RECV_DATA6 := FALSE;
   RECV8_DATA.RECV_DATA7 := FALSE;
   RECV8_DATA.RECV_DATA8 := FALSE;
   RECV8_DATA.RECV_STATUS := W#16#0;
   RECV8_DATA.RECV_LEN := 0;
   RECV8_DATA.SPARE2[0] := B#16#0;
   RECV8_DATA.SPARE2[1] := B#16#0;
   RECV8_DATA.SPARE2[2] := B#16#0;
   RECV8_DATA.SPARE2[3] := B#16#0;
   RECV9_DATA.RECV_NDR := FALSE;
   RECV9_DATA.RECV_ERROR := FALSE;
   RECV9_DATA.RECV_DATA3 := FALSE;
   RECV9_DATA.RECV_DATA4 := FALSE;
   RECV9_DATA.RECV_DATA5 := FALSE;
   RECV9_DATA.RECV_DATA6 := FALSE;
   RECV9_DATA.RECV_DATA7 := FALSE;
   RECV9_DATA.RECV_DATA8 := FALSE;
   RECV9_DATA.RECV_STATUS := W#16#0;
   RECV9_DATA.RECV_LEN := 0;
   RECV9_DATA.SPARE2[0] := B#16#0;
   RECV9_DATA.SPARE2[1] := B#16#0;
   RECV9_DATA.SPARE2[2] := B#16#0;
   RECV9_DATA.SPARE2[3] := B#16#0;
   RECV10_DATA.RECV_NDR := FALSE;
   RECV10_DATA.RECV_ERROR := FALSE;
   RECV10_DATA.RECV_DATA3 := FALSE;
   RECV10_DATA.RECV_DATA4 := FALSE;
   RECV10_DATA.RECV_DATA5 := FALSE;
   RECV10_DATA.RECV_DATA6 := FALSE;
   RECV10_DATA.RECV_DATA7 := FALSE;
   RECV10_DATA.RECV_DATA8 := FALSE;
   RECV10_DATA.RECV_STATUS := W#16#0;
   RECV10_DATA.RECV_LEN := 0;
   RECV10_DATA.SPARE2[0] := B#16#0;
   RECV10_DATA.SPARE2[1] := B#16#0;
   RECV10_DATA.SPARE2[2] := B#16#0;
   RECV10_DATA.SPARE2[3] := B#16#0;
   SEND11_DATA.SEND_DONE := FALSE;
   SEND11_DATA.SEND_ERROR := FALSE;
   SEND11_DATA.SEND_SCAN := FALSE;
   SEND11_DATA.SEND_ACT := FALSE;
   SEND11_DATA.SEND_SP1 := FALSE;
   SEND11_DATA.SEND_SP2 := FALSE;
   SEND11_DATA.SEND_SP3 := FALSE;
   SEND11_DATA.SEND_SP4 := FALSE;
   SEND11_DATA.SEND_STATUS := W#16#0;
   SEND11_DATA.SPARE2[0] := W#16#0;
   SEND11_DATA.SPARE2[1] := W#16#0;
   SEND11_DATA.SPARE2[2] := W#16#0;
   SEND12_DATA.SEND_DONE := FALSE;
   SEND12_DATA.SEND_ERROR := FALSE;
   SEND12_DATA.SEND_SCAN := FALSE;
   SEND12_DATA.SEND_ACT := FALSE;
   SEND12_DATA.SEND_SP1 := FALSE;
   SEND12_DATA.SEND_SP2 := FALSE;
   SEND12_DATA.SEND_SP3 := FALSE;
   SEND12_DATA.SEND_SP4 := FALSE;
   SEND12_DATA.SEND_STATUS := W#16#0;
   SEND12_DATA.SPARE2[0] := W#16#0;
   SEND12_DATA.SPARE2[1] := W#16#0;
   SEND12_DATA.SPARE2[2] := W#16#0;
   SEND13_DATA.SEND_DONE := FALSE;
   SEND13_DATA.SEND_ERROR := FALSE;
   SEND13_DATA.SEND_SCAN := FALSE;
   SEND13_DATA.SEND_ACT := FALSE;
   SEND13_DATA.SEND_SP1 := FALSE;
   SEND13_DATA.SEND_SP2 := FALSE;
   SEND13_DATA.SEND_SP3 := FALSE;
   SEND13_DATA.SEND_SP4 := FALSE;
   SEND13_DATA.SEND_STATUS := W#16#0;
   SEND13_DATA.SPARE2[0] := W#16#0;
   SEND13_DATA.SPARE2[1] := W#16#0;
   SEND13_DATA.SPARE2[2] := W#16#0;
   SEND14_DATA.SEND_DONE := FALSE;
   SEND14_DATA.SEND_ERROR := FALSE;
   SEND14_DATA.SEND_SCAN := FALSE;
   SEND14_DATA.SEND_ACT := FALSE;
   SEND14_DATA.SEND_SP1 := FALSE;
   SEND14_DATA.SEND_SP2 := FALSE;
   SEND14_DATA.SEND_SP3 := FALSE;
   SEND14_DATA.SEND_SP4 := FALSE;
   SEND14_DATA.SEND_STATUS := W#16#0;
   SEND14_DATA.SPARE2[0] := W#16#0;
   SEND14_DATA.SPARE2[1] := W#16#0;
   SEND14_DATA.SPARE2[2] := W#16#0;
   SEND15_DATA.SEND_DONE := FALSE;
   SEND15_DATA.SEND_ERROR := FALSE;
   SEND15_DATA.SEND_SCAN := FALSE;
   SEND15_DATA.SEND_ACT := FALSE;
   SEND15_DATA.SEND_SP1 := FALSE;
   SEND15_DATA.SEND_SP2 := FALSE;
   SEND15_DATA.SEND_SP3 := FALSE;
   SEND15_DATA.SEND_SP4 := FALSE;
   SEND15_DATA.SEND_STATUS := W#16#0;
   SEND15_DATA.SPARE2[0] := W#16#0;
   SEND15_DATA.SPARE2[1] := W#16#0;
   SEND15_DATA.SPARE2[2] := W#16#0;
   SEND16_DATA.SEND_DONE := FALSE;
   SEND16_DATA.SEND_ERROR := FALSE;
   SEND16_DATA.SEND_SCAN := FALSE;
   SEND16_DATA.SEND_ACT := FALSE;
   SEND16_DATA.SEND_SP1 := FALSE;
   SEND16_DATA.SEND_SP2 := FALSE;
   SEND16_DATA.SEND_SP3 := FALSE;
   SEND16_DATA.SEND_SP4 := FALSE;
   SEND16_DATA.SEND_STATUS := W#16#0;
   SEND16_DATA.SPARE2[0] := W#16#0;
   SEND16_DATA.SPARE2[1] := W#16#0;
   SEND16_DATA.SPARE2[2] := W#16#0;
   SEND17_DATA.SEND_DONE := FALSE;
   SEND17_DATA.SEND_ERROR := FALSE;
   SEND17_DATA.SEND_SCAN := FALSE;
   SEND17_DATA.SEND_ACT := FALSE;
   SEND17_DATA.SEND_SP1 := FALSE;
   SEND17_DATA.SEND_SP2 := FALSE;
   SEND17_DATA.SEND_SP3 := FALSE;
   SEND17_DATA.SEND_SP4 := FALSE;
   SEND17_DATA.SEND_STATUS := W#16#0;
   SEND17_DATA.SPARE2[0] := W#16#0;
   SEND17_DATA.SPARE2[1] := W#16#0;
   SEND17_DATA.SPARE2[2] := W#16#0;
   SEND18_DATA.SEND_DONE := FALSE;
   SEND18_DATA.SEND_ERROR := FALSE;
   SEND18_DATA.SEND_SCAN := FALSE;
   SEND18_DATA.SEND_ACT := FALSE;
   SEND18_DATA.SEND_SP1 := FALSE;
   SEND18_DATA.SEND_SP2 := FALSE;
   SEND18_DATA.SEND_SP3 := FALSE;
   SEND18_DATA.SEND_SP4 := FALSE;
   SEND18_DATA.SEND_STATUS := W#16#0;
   SEND18_DATA.SPARE2[0] := W#16#0;
   SEND18_DATA.SPARE2[1] := W#16#0;
   SEND18_DATA.SPARE2[2] := W#16#0;
   SEND19_DATA.SEND_DONE := FALSE;
   SEND19_DATA.SEND_ERROR := FALSE;
   SEND19_DATA.SEND_SCAN := FALSE;
   SEND19_DATA.SEND_ACT := FALSE;
   SEND19_DATA.SEND_SP1 := FALSE;
   SEND19_DATA.SEND_SP2 := FALSE;
   SEND19_DATA.SEND_SP3 := FALSE;
   SEND19_DATA.SEND_SP4 := FALSE;
   SEND19_DATA.SEND_STATUS := W#16#0;
   SEND19_DATA.SPARE2[0] := W#16#0;
   SEND19_DATA.SPARE2[1] := W#16#0;
   SEND19_DATA.SPARE2[2] := W#16#0;
   SEND20_DATA.SEND_DONE := FALSE;
   SEND20_DATA.SEND_ERROR := FALSE;
   SEND20_DATA.SEND_SCAN := FALSE;
   SEND20_DATA.SEND_ACT := FALSE;
   SEND20_DATA.SEND_SP1 := FALSE;
   SEND20_DATA.SEND_SP2 := FALSE;
   SEND20_DATA.SEND_SP3 := FALSE;
   SEND20_DATA.SEND_SP4 := FALSE;
   SEND20_DATA.SEND_STATUS := W#16#0;
   SEND20_DATA.SPARE2[0] := W#16#0;
   SEND20_DATA.SPARE2[1] := W#16#0;
   SEND20_DATA.SPARE2[2] := W#16#0;
   RECV11_DATA.RECV_NDR := FALSE;
   RECV11_DATA.RECV_ERROR := FALSE;
   RECV11_DATA.RECV_DATA3 := FALSE;
   RECV11_DATA.RECV_DATA4 := FALSE;
   RECV11_DATA.RECV_DATA5 := FALSE;
   RECV11_DATA.RECV_DATA6 := FALSE;
   RECV11_DATA.RECV_DATA7 := FALSE;
   RECV11_DATA.RECV_DATA8 := FALSE;
   RECV11_DATA.RECV_STATUS := W#16#0;
   RECV11_DATA.RECV_LEN := 0;
   RECV11_DATA.SPARE2[0] := B#16#0;
   RECV11_DATA.SPARE2[1] := B#16#0;
   RECV11_DATA.SPARE2[2] := B#16#0;
   RECV11_DATA.SPARE2[3] := B#16#0;
   RECV12_DATA.RECV_NDR := FALSE;
   RECV12_DATA.RECV_ERROR := FALSE;
   RECV12_DATA.RECV_DATA3 := FALSE;
   RECV12_DATA.RECV_DATA4 := FALSE;
   RECV12_DATA.RECV_DATA5 := FALSE;
   RECV12_DATA.RECV_DATA6 := FALSE;
   RECV12_DATA.RECV_DATA7 := FALSE;
   RECV12_DATA.RECV_DATA8 := FALSE;
   RECV12_DATA.RECV_STATUS := W#16#0;
   RECV12_DATA.RECV_LEN := 0;
   RECV12_DATA.SPARE2[0] := B#16#0;
   RECV12_DATA.SPARE2[1] := B#16#0;
   RECV12_DATA.SPARE2[2] := B#16#0;
   RECV12_DATA.SPARE2[3] := B#16#0;
   RECV13_DATA.RECV_NDR := FALSE;
   RECV13_DATA.RECV_ERROR := FALSE;
   RECV13_DATA.RECV_DATA3 := FALSE;
   RECV13_DATA.RECV_DATA4 := FALSE;
   RECV13_DATA.RECV_DATA5 := FALSE;
   RECV13_DATA.RECV_DATA6 := FALSE;
   RECV13_DATA.RECV_DATA7 := FALSE;
   RECV13_DATA.RECV_DATA8 := FALSE;
   RECV13_DATA.RECV_STATUS := W#16#0;
   RECV13_DATA.RECV_LEN := 0;
   RECV13_DATA.SPARE2[0] := B#16#0;
   RECV13_DATA.SPARE2[1] := B#16#0;
   RECV13_DATA.SPARE2[2] := B#16#0;
   RECV13_DATA.SPARE2[3] := B#16#0;
   RECV14_DATA.RECV_NDR := FALSE;
   RECV14_DATA.RECV_ERROR := FALSE;
   RECV14_DATA.RECV_DATA3 := FALSE;
   RECV14_DATA.RECV_DATA4 := FALSE;
   RECV14_DATA.RECV_DATA5 := FALSE;
   RECV14_DATA.RECV_DATA6 := FALSE;
   RECV14_DATA.RECV_DATA7 := FALSE;
   RECV14_DATA.RECV_DATA8 := FALSE;
   RECV14_DATA.RECV_STATUS := W#16#0;
   RECV14_DATA.RECV_LEN := 0;
   RECV14_DATA.SPARE2[0] := B#16#0;
   RECV14_DATA.SPARE2[1] := B#16#0;
   RECV14_DATA.SPARE2[2] := B#16#0;
   RECV14_DATA.SPARE2[3] := B#16#0;
   RECV15_DATA.RECV_NDR := FALSE;
   RECV15_DATA.RECV_ERROR := FALSE;
   RECV15_DATA.RECV_DATA3 := FALSE;
   RECV15_DATA.RECV_DATA4 := FALSE;
   RECV15_DATA.RECV_DATA5 := FALSE;
   RECV15_DATA.RECV_DATA6 := FALSE;
   RECV15_DATA.RECV_DATA7 := FALSE;
   RECV15_DATA.RECV_DATA8 := FALSE;
   RECV15_DATA.RECV_STATUS := W#16#0;
   RECV15_DATA.RECV_LEN := 0;
   RECV15_DATA.SPARE2[0] := B#16#0;
   RECV15_DATA.SPARE2[1] := B#16#0;
   RECV15_DATA.SPARE2[2] := B#16#0;
   RECV15_DATA.SPARE2[3] := B#16#0;
   RECV16_DATA.RECV_NDR := FALSE;
   RECV16_DATA.RECV_ERROR := FALSE;
   RECV16_DATA.RECV_DATA3 := FALSE;
   RECV16_DATA.RECV_DATA4 := FALSE;
   RECV16_DATA.RECV_DATA5 := FALSE;
   RECV16_DATA.RECV_DATA6 := FALSE;
   RECV16_DATA.RECV_DATA7 := FALSE;
   RECV16_DATA.RECV_DATA8 := FALSE;
   RECV16_DATA.RECV_STATUS := W#16#0;
   RECV16_DATA.RECV_LEN := 0;
   RECV16_DATA.SPARE2[0] := B#16#0;
   RECV16_DATA.SPARE2[1] := B#16#0;
   RECV16_DATA.SPARE2[2] := B#16#0;
   RECV16_DATA.SPARE2[3] := B#16#0;
   RECV17_DATA.RECV_NDR := FALSE;
   RECV17_DATA.RECV_ERROR := FALSE;
   RECV17_DATA.RECV_DATA3 := FALSE;
   RECV17_DATA.RECV_DATA4 := FALSE;
   RECV17_DATA.RECV_DATA5 := FALSE;
   RECV17_DATA.RECV_DATA6 := FALSE;
   RECV17_DATA.RECV_DATA7 := FALSE;
   RECV17_DATA.RECV_DATA8 := FALSE;
   RECV17_DATA.RECV_STATUS := W#16#0;
   RECV17_DATA.RECV_LEN := 0;
   RECV17_DATA.SPARE2[0] := B#16#0;
   RECV17_DATA.SPARE2[1] := B#16#0;
   RECV17_DATA.SPARE2[2] := B#16#0;
   RECV17_DATA.SPARE2[3] := B#16#0;
   RECV18_DATA.RECV_NDR := FALSE;
   RECV18_DATA.RECV_ERROR := FALSE;
   RECV18_DATA.RECV_DATA3 := FALSE;
   RECV18_DATA.RECV_DATA4 := FALSE;
   RECV18_DATA.RECV_DATA5 := FALSE;
   RECV18_DATA.RECV_DATA6 := FALSE;
   RECV18_DATA.RECV_DATA7 := FALSE;
   RECV18_DATA.RECV_DATA8 := FALSE;
   RECV18_DATA.RECV_STATUS := W#16#0;
   RECV18_DATA.RECV_LEN := 0;
   RECV18_DATA.SPARE2[0] := B#16#0;
   RECV18_DATA.SPARE2[1] := B#16#0;
   RECV18_DATA.SPARE2[2] := B#16#0;
   RECV18_DATA.SPARE2[3] := B#16#0;
   RECV19_DATA.RECV_NDR := FALSE;
   RECV19_DATA.RECV_ERROR := FALSE;
   RECV19_DATA.RECV_DATA3 := FALSE;
   RECV19_DATA.RECV_DATA4 := FALSE;
   RECV19_DATA.RECV_DATA5 := FALSE;
   RECV19_DATA.RECV_DATA6 := FALSE;
   RECV19_DATA.RECV_DATA7 := FALSE;
   RECV19_DATA.RECV_DATA8 := FALSE;
   RECV19_DATA.RECV_STATUS := W#16#0;
   RECV19_DATA.RECV_LEN := 0;
   RECV19_DATA.SPARE2[0] := B#16#0;
   RECV19_DATA.SPARE2[1] := B#16#0;
   RECV19_DATA.SPARE2[2] := B#16#0;
   RECV19_DATA.SPARE2[3] := B#16#0;
   RECV20_DATA.RECV_NDR := FALSE;
   RECV20_DATA.RECV_ERROR := FALSE;
   RECV20_DATA.RECV_DATA3 := FALSE;
   RECV20_DATA.RECV_DATA4 := FALSE;
   RECV20_DATA.RECV_DATA5 := FALSE;
   RECV20_DATA.RECV_DATA6 := FALSE;
   RECV20_DATA.RECV_DATA7 := FALSE;
   RECV20_DATA.RECV_DATA8 := FALSE;
   RECV20_DATA.RECV_STATUS := W#16#0;
   RECV20_DATA.RECV_LEN := 0;
   RECV20_DATA.SPARE2[0] := B#16#0;
   RECV20_DATA.SPARE2[1] := B#16#0;
   RECV20_DATA.SPARE2[2] := B#16#0;
   RECV20_DATA.SPARE2[3] := B#16#0;
END_DATA_BLOCK

DATA_BLOCK DB 18
TITLE =
VERSION : 0.1


  STRUCT
   SHUTTLE : STRUCT 	//Temporary placeholder variable
    DATA1 : WORD ;
    DATA2 : WORD ;
    DATA3 : WORD ;
    DATA4 : WORD ;
    DATA5 : WORD ;
    DATA6 : WORD ;
    DATA7 : WORD ;
    DATA8 : WORD ;
    DATA9 : WORD ;
    DATA10 : WORD ;
   END_STRUCT ;
   S481 : STRUCT 	//Temporary placeholder variable
    DATA1 : WORD ;
    DATA2 : WORD ;
    DATA3 : WORD ;
    DATA4 : WORD ;
    DATA5 : WORD ;
    DATA6 : WORD ;
    DATA7 : WORD ;
    DATA8 : WORD ;
    DATA9 : WORD ;
    DATA10 : WORD ;
   END_STRUCT ;
   S482 : STRUCT 	//Temporary placeholder variable
    DATA1 : WORD ;
    DATA2 : WORD ;
    DATA3 : WORD ;
    DATA4 : WORD ;
    DATA5 : WORD ;
    DATA6 : WORD ;
    DATA7 : WORD ;
    DATA8 : WORD ;
    DATA9 : WORD ;
    DATA10 : WORD ;
   END_STRUCT ;
   S483 : STRUCT 	//Temporary placeholder variable
    DATA1 : WORD ;
    DATA2 : WORD ;
    DATA3 : WORD ;
    DATA4 : WORD ;
    DATA5 : WORD ;
    DATA6 : WORD ;
    DATA7 : WORD ;
    DATA8 : WORD ;
    DATA9 : WORD ;
    DATA10 : WORD ;
   END_STRUCT ;
   SPARE1 : STRUCT 	//Temporary placeholder variable
    DATA1 : WORD ;
    DATA2 : WORD ;
    DATA3 : WORD ;
    DATA4 : WORD ;
    DATA5 : WORD ;
    DATA6 : WORD ;
    DATA7 : WORD ;
    DATA8 : WORD ;
    DATA9 : WORD ;
    DATA10 : WORD ;
   END_STRUCT ;
   SPARE2 : STRUCT 	//Temporary placeholder variable
    DATA1 : WORD ;
    DATA2 : WORD ;
    DATA3 : WORD ;
    DATA4 : WORD ;
    DATA5 : WORD ;
    DATA6 : WORD ;
    DATA7 : WORD ;
    DATA8 : WORD ;
    DATA9 : WORD ;
    DATA10 : WORD ;
   END_STRUCT ;
   SPARE3 : STRUCT 	//Temporary placeholder variable
    DATA1 : WORD ;
    DATA2 : WORD ;
    DATA3 : WORD ;
    DATA4 : WORD ;
    DATA5 : WORD ;
    DATA6 : WORD ;
    DATA7 : WORD ;
    DATA8 : WORD ;
    DATA9 : WORD ;
    DATA10 : WORD ;
   END_STRUCT ;
   SPARE4 : STRUCT 	//Temporary placeholder variable
    DATA1 : WORD ;
    DATA2 : WORD ;
    DATA3 : WORD ;
    DATA4 : WORD ;
    DATA5 : WORD ;
    DATA6 : WORD ;
    DATA7 : WORD ;
    DATA8 : WORD ;
    DATA9 : WORD ;
    DATA10 : WORD ;
   END_STRUCT ;
   SPARE5 : STRUCT 	//Temporary placeholder variable
    DATA1 : WORD ;
    DATA2 : WORD ;
    DATA3 : WORD ;
    DATA4 : WORD ;
    DATA5 : WORD ;
    DATA6 : WORD ;
    DATA7 : WORD ;
    DATA8 : WORD ;
    DATA9 : WORD ;
    DATA10 : WORD ;
   END_STRUCT ;
   SPARE6 : STRUCT 	//Temporary placeholder variable
    DATA1 : WORD ;
    DATA2 : WORD ;
    DATA3 : WORD ;
    DATA4 : WORD ;
    DATA5 : WORD ;
    DATA6 : WORD ;
    DATA7 : WORD ;
    DATA8 : WORD ;
    DATA9 : WORD ;
    DATA10 : WORD ;
   END_STRUCT ;
  END_STRUCT ;
BEGIN
   SHUTTLE.DATA1 := W#16#0;
   SHUTTLE.DATA2 := W#16#0;
   SHUTTLE.DATA3 := W#16#0;
   SHUTTLE.DATA4 := W#16#0;
   SHUTTLE.DATA5 := W#16#0;
   SHUTTLE.DATA6 := W#16#0;
   SHUTTLE.DATA7 := W#16#0;
   SHUTTLE.DATA8 := W#16#0;
   SHUTTLE.DATA9 := W#16#0;
   SHUTTLE.DATA10 := W#16#0;
   S481.DATA1 := W#16#0;
   S481.DATA2 := W#16#0;
   S481.DATA3 := W#16#0;
   S481.DATA4 := W#16#0;
   S481.DATA5 := W#16#0;
   S481.DATA6 := W#16#0;
   S481.DATA7 := W#16#0;
   S481.DATA8 := W#16#0;
   S481.DATA9 := W#16#0;
   S481.DATA10 := W#16#0;
   S482.DATA1 := W#16#0;
   S482.DATA2 := W#16#0;
   S482.DATA3 := W#16#0;
   S482.DATA4 := W#16#0;
   S482.DATA5 := W#16#0;
   S482.DATA6 := W#16#0;
   S482.DATA7 := W#16#0;
   S482.DATA8 := W#16#0;
   S482.DATA9 := W#16#0;
   S482.DATA10 := W#16#0;
   S483.DATA1 := W#16#0;
   S483.DATA2 := W#16#0;
   S483.DATA3 := W#16#0;
   S483.DATA4 := W#16#0;
   S483.DATA5 := W#16#0;
   S483.DATA6 := W#16#0;
   S483.DATA7 := W#16#0;
   S483.DATA8 := W#16#0;
   S483.DATA9 := W#16#0;
   S483.DATA10 := W#16#0;
   SPARE1.DATA1 := W#16#0;
   SPARE1.DATA2 := W#16#0;
   SPARE1.DATA3 := W#16#0;
   SPARE1.DATA4 := W#16#0;
   SPARE1.DATA5 := W#16#0;
   SPARE1.DATA6 := W#16#0;
   SPARE1.DATA7 := W#16#0;
   SPARE1.DATA8 := W#16#0;
   SPARE1.DATA9 := W#16#0;
   SPARE1.DATA10 := W#16#0;
   SPARE2.DATA1 := W#16#0;
   SPARE2.DATA2 := W#16#0;
   SPARE2.DATA3 := W#16#0;
   SPARE2.DATA4 := W#16#0;
   SPARE2.DATA5 := W#16#0;
   SPARE2.DATA6 := W#16#0;
   SPARE2.DATA7 := W#16#0;
   SPARE2.DATA8 := W#16#0;
   SPARE2.DATA9 := W#16#0;
   SPARE2.DATA10 := W#16#0;
   SPARE3.DATA1 := W#16#0;
   SPARE3.DATA2 := W#16#0;
   SPARE3.DATA3 := W#16#0;
   SPARE3.DATA4 := W#16#0;
   SPARE3.DATA5 := W#16#0;
   SPARE3.DATA6 := W#16#0;
   SPARE3.DATA7 := W#16#0;
   SPARE3.DATA8 := W#16#0;
   SPARE3.DATA9 := W#16#0;
   SPARE3.DATA10 := W#16#0;
   SPARE4.DATA1 := W#16#0;
   SPARE4.DATA2 := W#16#0;
   SPARE4.DATA3 := W#16#0;
   SPARE4.DATA4 := W#16#0;
   SPARE4.DATA5 := W#16#0;
   SPARE4.DATA6 := W#16#0;
   SPARE4.DATA7 := W#16#0;
   SPARE4.DATA8 := W#16#0;
   SPARE4.DATA9 := W#16#0;
   SPARE4.DATA10 := W#16#0;
   SPARE5.DATA1 := W#16#0;
   SPARE5.DATA2 := W#16#0;
   SPARE5.DATA3 := W#16#0;
   SPARE5.DATA4 := W#16#0;
   SPARE5.DATA5 := W#16#0;
   SPARE5.DATA6 := W#16#0;
   SPARE5.DATA7 := W#16#0;
   SPARE5.DATA8 := W#16#0;
   SPARE5.DATA9 := W#16#0;
   SPARE5.DATA10 := W#16#0;
   SPARE6.DATA1 := W#16#0;
   SPARE6.DATA2 := W#16#0;
   SPARE6.DATA3 := W#16#0;
   SPARE6.DATA4 := W#16#0;
   SPARE6.DATA5 := W#16#0;
   SPARE6.DATA6 := W#16#0;
   SPARE6.DATA7 := W#16#0;
   SPARE6.DATA8 := W#16#0;
   SPARE6.DATA9 := W#16#0;
   SPARE6.DATA10 := W#16#0;
END_DATA_BLOCK

DATA_BLOCK DB 28
TITLE =
VERSION : 0.1


  STRUCT
   SPARE1 : STRUCT 	//Temporary placeholder variable
    DATA1 : WORD ;
    DATA2 : WORD ;
    DATA3 : WORD ;
    DATA4 : WORD ;
    DATA5 : WORD ;
    DATA6 : WORD ;
    DATA7 : WORD ;
    DATA8 : WORD ;
    DATA9 : WORD ;
    DATA10 : WORD ;
   END_STRUCT ;
   SPARE2 : STRUCT 	//Temporary placeholder variable
    DATA1 : WORD ;
    DATA2 : WORD ;
    DATA3 : WORD ;
    DATA4 : WORD ;
    DATA5 : WORD ;
    DATA6 : WORD ;
    DATA7 : WORD ;
    DATA8 : WORD ;
    DATA9 : WORD ;
    DATA10 : WORD ;
   END_STRUCT ;
   SPARE3 : STRUCT 	//Temporary placeholder variable
    DATA1 : WORD ;
    DATA2 : WORD ;
    DATA3 : WORD ;
    DATA4 : WORD ;
    DATA5 : WORD ;
    DATA6 : WORD ;
    DATA7 : WORD ;
    DATA8 : WORD ;
    DATA9 : WORD ;
    DATA10 : WORD ;
   END_STRUCT ;
   SPARE4 : STRUCT 	//Temporary placeholder variable
    DATA1 : WORD ;
    DATA2 : WORD ;
    DATA3 : WORD ;
    DATA4 : WORD ;
    DATA5 : WORD ;
    DATA6 : WORD ;
    DATA7 : WORD ;
    DATA8 : WORD ;
    DATA9 : WORD ;
    DATA10 : WORD ;
   END_STRUCT ;
   S484 : STRUCT 	//Temporary placeholder variable
    DATA1 : WORD ;
    DATA2 : WORD ;
    DATA3 : WORD ;
    DATA4 : WORD ;
    DATA5 : WORD ;
    DATA6 : WORD ;
    DATA7 : WORD ;
    DATA8 : WORD ;
    DATA9 : WORD ;
    DATA10 : WORD ;
   END_STRUCT ;
   S485 : STRUCT 	//Temporary placeholder variable
    DATA1 : WORD ;
    DATA2 : WORD ;
    DATA3 : WORD ;
    DATA4 : WORD ;
    DATA5 : WORD ;
    DATA6 : WORD ;
    DATA7 : WORD ;
    DATA8 : WORD ;
    DATA9 : WORD ;
    DATA10 : WORD ;
   END_STRUCT ;
   S486 : STRUCT 	//Temporary placeholder variable
    DATA1 : WORD ;
    DATA2 : WORD ;
    DATA3 : WORD ;
    DATA4 : WORD ;
    DATA5 : WORD ;
    DATA6 : WORD ;
    DATA7 : WORD ;
    DATA8 : WORD ;
    DATA9 : WORD ;
    DATA10 : WORD ;
   END_STRUCT ;
   S487_8 : STRUCT 	//Temporary placeholder variable
    DATA1 : WORD ;
    DATA2 : WORD ;
    DATA3 : WORD ;
    DATA4 : WORD ;
    DATA5 : WORD ;
    DATA6 : WORD ;
    DATA7 : WORD ;
    DATA8 : WORD ;
    DATA9 : WORD ;
    DATA10 : WORD ;
   END_STRUCT ;
   SPARE5 : STRUCT 	//Temporary placeholder variable
    DATA1 : WORD ;
    DATA2 : WORD ;
    DATA3 : WORD ;
    DATA4 : WORD ;
    DATA5 : WORD ;
    DATA6 : WORD ;
    DATA7 : WORD ;
    DATA8 : WORD ;
    DATA9 : WORD ;
    DATA10 : WORD ;
   END_STRUCT ;
   SPARE6 : STRUCT 	//Temporary placeholder variable
    DATA1 : WORD ;
    DATA2 : WORD ;
    DATA3 : WORD ;
    DATA4 : WORD ;
    DATA5 : WORD ;
    DATA6 : WORD ;
    DATA7 : WORD ;
    DATA8 : WORD ;
    DATA9 : WORD ;
    DATA10 : WORD ;
   END_STRUCT ;
  END_STRUCT ;
BEGIN
   SPARE1.DATA1 := W#16#0;
   SPARE1.DATA2 := W#16#0;
   SPARE1.DATA3 := W#16#0;
   SPARE1.DATA4 := W#16#0;
   SPARE1.DATA5 := W#16#0;
   SPARE1.DATA6 := W#16#0;
   SPARE1.DATA7 := W#16#0;
   SPARE1.DATA8 := W#16#0;
   SPARE1.DATA9 := W#16#0;
   SPARE1.DATA10 := W#16#0;
   SPARE2.DATA1 := W#16#0;
   SPARE2.DATA2 := W#16#0;
   SPARE2.DATA3 := W#16#0;
   SPARE2.DATA4 := W#16#0;
   SPARE2.DATA5 := W#16#0;
   SPARE2.DATA6 := W#16#0;
   SPARE2.DATA7 := W#16#0;
   SPARE2.DATA8 := W#16#0;
   SPARE2.DATA9 := W#16#0;
   SPARE2.DATA10 := W#16#0;
   SPARE3.DATA1 := W#16#0;
   SPARE3.DATA2 := W#16#0;
   SPARE3.DATA3 := W#16#0;
   SPARE3.DATA4 := W#16#0;
   SPARE3.DATA5 := W#16#0;
   SPARE3.DATA6 := W#16#0;
   SPARE3.DATA7 := W#16#0;
   SPARE3.DATA8 := W#16#0;
   SPARE3.DATA9 := W#16#0;
   SPARE3.DATA10 := W#16#0;
   SPARE4.DATA1 := W#16#0;
   SPARE4.DATA2 := W#16#0;
   SPARE4.DATA3 := W#16#0;
   SPARE4.DATA4 := W#16#0;
   SPARE4.DATA5 := W#16#0;
   SPARE4.DATA6 := W#16#0;
   SPARE4.DATA7 := W#16#0;
   SPARE4.DATA8 := W#16#0;
   SPARE4.DATA9 := W#16#0;
   SPARE4.DATA10 := W#16#0;
   S484.DATA1 := W#16#0;
   S484.DATA2 := W#16#0;
   S484.DATA3 := W#16#0;
   S484.DATA4 := W#16#0;
   S484.DATA5 := W#16#0;
   S484.DATA6 := W#16#0;
   S484.DATA7 := W#16#0;
   S484.DATA8 := W#16#0;
   S484.DATA9 := W#16#0;
   S484.DATA10 := W#16#0;
   S485.DATA1 := W#16#0;
   S485.DATA2 := W#16#0;
   S485.DATA3 := W#16#0;
   S485.DATA4 := W#16#0;
   S485.DATA5 := W#16#0;
   S485.DATA6 := W#16#0;
   S485.DATA7 := W#16#0;
   S485.DATA8 := W#16#0;
   S485.DATA9 := W#16#0;
   S485.DATA10 := W#16#0;
   S486.DATA1 := W#16#0;
   S486.DATA2 := W#16#0;
   S486.DATA3 := W#16#0;
   S486.DATA4 := W#16#0;
   S486.DATA5 := W#16#0;
   S486.DATA6 := W#16#0;
   S486.DATA7 := W#16#0;
   S486.DATA8 := W#16#0;
   S486.DATA9 := W#16#0;
   S486.DATA10 := W#16#0;
   S487_8.DATA1 := W#16#0;
   S487_8.DATA2 := W#16#0;
   S487_8.DATA3 := W#16#0;
   S487_8.DATA4 := W#16#0;
   S487_8.DATA5 := W#16#0;
   S487_8.DATA6 := W#16#0;
   S487_8.DATA7 := W#16#0;
   S487_8.DATA8 := W#16#0;
   S487_8.DATA9 := W#16#0;
   S487_8.DATA10 := W#16#0;
   SPARE5.DATA1 := W#16#0;
   SPARE5.DATA2 := W#16#0;
   SPARE5.DATA3 := W#16#0;
   SPARE5.DATA4 := W#16#0;
   SPARE5.DATA5 := W#16#0;
   SPARE5.DATA6 := W#16#0;
   SPARE5.DATA7 := W#16#0;
   SPARE5.DATA8 := W#16#0;
   SPARE5.DATA9 := W#16#0;
   SPARE5.DATA10 := W#16#0;
   SPARE6.DATA1 := W#16#0;
   SPARE6.DATA2 := W#16#0;
   SPARE6.DATA3 := W#16#0;
   SPARE6.DATA4 := W#16#0;
   SPARE6.DATA5 := W#16#0;
   SPARE6.DATA6 := W#16#0;
   SPARE6.DATA7 := W#16#0;
   SPARE6.DATA8 := W#16#0;
   SPARE6.DATA9 := W#16#0;
   SPARE6.DATA10 := W#16#0;
END_DATA_BLOCK

DATA_BLOCK DB 50
TITLE =
VERSION : 0.1


  STRUCT
   STAT0 : ARRAY  [0 .. 255 ] OF //G.P DATA BLOCK
   WORD  := W#16#0;
  END_STRUCT ;
BEGIN
   STAT0[0] := W#16#0;
   STAT0[1] := W#16#0;
   STAT0[2] := W#16#0;
   STAT0[3] := W#16#0;
   STAT0[4] := W#16#0;
   STAT0[5] := W#16#0;
   STAT0[6] := W#16#0;
   STAT0[7] := W#16#0;
   STAT0[8] := W#16#0;
   STAT0[9] := W#16#0;
   STAT0[10] := W#16#0;
   STAT0[11] := W#16#0;
   STAT0[12] := W#16#0;
   STAT0[13] := W#16#0;
   STAT0[14] := W#16#0;
   STAT0[15] := W#16#0;
   STAT0[16] := W#16#0;
   STAT0[17] := W#16#0;
   STAT0[18] := W#16#0;
   STAT0[19] := W#16#0;
   STAT0[20] := W#16#0;
   STAT0[21] := W#16#0;
   STAT0[22] := W#16#0;
   STAT0[23] := W#16#0;
   STAT0[24] := W#16#0;
   STAT0[25] := W#16#0;
   STAT0[26] := W#16#0;
   STAT0[27] := W#16#0;
   STAT0[28] := W#16#0;
   STAT0[29] := W#16#0;
   STAT0[30] := W#16#0;
   STAT0[31] := W#16#0;
   STAT0[32] := W#16#0;
   STAT0[33] := W#16#0;
   STAT0[34] := W#16#0;
   STAT0[35] := W#16#0;
   STAT0[36] := W#16#0;
   STAT0[37] := W#16#0;
   STAT0[38] := W#16#0;
   STAT0[39] := W#16#0;
   STAT0[40] := W#16#0;
   STAT0[41] := W#16#0;
   STAT0[42] := W#16#0;
   STAT0[43] := W#16#0;
   STAT0[44] := W#16#0;
   STAT0[45] := W#16#0;
   STAT0[46] := W#16#0;
   STAT0[47] := W#16#0;
   STAT0[48] := W#16#0;
   STAT0[49] := W#16#0;
   STAT0[50] := W#16#0;
   STAT0[51] := W#16#0;
   STAT0[52] := W#16#0;
   STAT0[53] := W#16#0;
   STAT0[54] := W#16#0;
   STAT0[55] := W#16#0;
   STAT0[56] := W#16#0;
   STAT0[57] := W#16#0;
   STAT0[58] := W#16#0;
   STAT0[59] := W#16#0;
   STAT0[60] := W#16#0;
   STAT0[61] := W#16#0;
   STAT0[62] := W#16#0;
   STAT0[63] := W#16#0;
   STAT0[64] := W#16#0;
   STAT0[65] := W#16#0;
   STAT0[66] := W#16#0;
   STAT0[67] := W#16#0;
   STAT0[68] := W#16#0;
   STAT0[69] := W#16#0;
   STAT0[70] := W#16#0;
   STAT0[71] := W#16#0;
   STAT0[72] := W#16#0;
   STAT0[73] := W#16#0;
   STAT0[74] := W#16#0;
   STAT0[75] := W#16#0;
   STAT0[76] := W#16#0;
   STAT0[77] := W#16#0;
   STAT0[78] := W#16#0;
   STAT0[79] := W#16#0;
   STAT0[80] := W#16#0;
   STAT0[81] := W#16#0;
   STAT0[82] := W#16#0;
   STAT0[83] := W#16#0;
   STAT0[84] := W#16#0;
   STAT0[85] := W#16#0;
   STAT0[86] := W#16#0;
   STAT0[87] := W#16#0;
   STAT0[88] := W#16#0;
   STAT0[89] := W#16#0;
   STAT0[90] := W#16#0;
   STAT0[91] := W#16#0;
   STAT0[92] := W#16#0;
   STAT0[93] := W#16#0;
   STAT0[94] := W#16#0;
   STAT0[95] := W#16#0;
   STAT0[96] := W#16#0;
   STAT0[97] := W#16#0;
   STAT0[98] := W#16#0;
   STAT0[99] := W#16#0;
   STAT0[100] := W#16#0;
   STAT0[101] := W#16#0;
   STAT0[102] := W#16#0;
   STAT0[103] := W#16#0;
   STAT0[104] := W#16#0;
   STAT0[105] := W#16#0;
   STAT0[106] := W#16#0;
   STAT0[107] := W#16#0;
   STAT0[108] := W#16#0;
   STAT0[109] := W#16#0;
   STAT0[110] := W#16#0;
   STAT0[111] := W#16#0;
   STAT0[112] := W#16#0;
   STAT0[113] := W#16#0;
   STAT0[114] := W#16#0;
   STAT0[115] := W#16#0;
   STAT0[116] := W#16#0;
   STAT0[117] := W#16#0;
   STAT0[118] := W#16#0;
   STAT0[119] := W#16#0;
   STAT0[120] := W#16#0;
   STAT0[121] := W#16#0;
   STAT0[122] := W#16#0;
   STAT0[123] := W#16#0;
   STAT0[124] := W#16#0;
   STAT0[125] := W#16#0;
   STAT0[126] := W#16#0;
   STAT0[127] := W#16#0;
   STAT0[128] := W#16#0;
   STAT0[129] := W#16#0;
   STAT0[130] := W#16#0;
   STAT0[131] := W#16#0;
   STAT0[132] := W#16#0;
   STAT0[133] := W#16#0;
   STAT0[134] := W#16#0;
   STAT0[135] := W#16#0;
   STAT0[136] := W#16#0;
   STAT0[137] := W#16#0;
   STAT0[138] := W#16#0;
   STAT0[139] := W#16#0;
   STAT0[140] := W#16#0;
   STAT0[141] := W#16#0;
   STAT0[142] := W#16#0;
   STAT0[143] := W#16#0;
   STAT0[144] := W#16#0;
   STAT0[145] := W#16#0;
   STAT0[146] := W#16#0;
   STAT0[147] := W#16#0;
   STAT0[148] := W#16#0;
   STAT0[149] := W#16#0;
   STAT0[150] := W#16#0;
   STAT0[151] := W#16#0;
   STAT0[152] := W#16#0;
   STAT0[153] := W#16#0;
   STAT0[154] := W#16#0;
   STAT0[155] := W#16#0;
   STAT0[156] := W#16#0;
   STAT0[157] := W#16#0;
   STAT0[158] := W#16#0;
   STAT0[159] := W#16#0;
   STAT0[160] := W#16#0;
   STAT0[161] := W#16#0;
   STAT0[162] := W#16#0;
   STAT0[163] := W#16#0;
   STAT0[164] := W#16#0;
   STAT0[165] := W#16#0;
   STAT0[166] := W#16#0;
   STAT0[167] := W#16#0;
   STAT0[168] := W#16#0;
   STAT0[169] := W#16#0;
   STAT0[170] := W#16#0;
   STAT0[171] := W#16#0;
   STAT0[172] := W#16#0;
   STAT0[173] := W#16#0;
   STAT0[174] := W#16#0;
   STAT0[175] := W#16#0;
   STAT0[176] := W#16#0;
   STAT0[177] := W#16#0;
   STAT0[178] := W#16#0;
   STAT0[179] := W#16#0;
   STAT0[180] := W#16#0;
   STAT0[181] := W#16#0;
   STAT0[182] := W#16#0;
   STAT0[183] := W#16#0;
   STAT0[184] := W#16#0;
   STAT0[185] := W#16#0;
   STAT0[186] := W#16#0;
   STAT0[187] := W#16#0;
   STAT0[188] := W#16#0;
   STAT0[189] := W#16#0;
   STAT0[190] := W#16#0;
   STAT0[191] := W#16#0;
   STAT0[192] := W#16#0;
   STAT0[193] := W#16#0;
   STAT0[194] := W#16#0;
   STAT0[195] := W#16#0;
   STAT0[196] := W#16#0;
   STAT0[197] := W#16#0;
   STAT0[198] := W#16#0;
   STAT0[199] := W#16#0;
   STAT0[200] := W#16#0;
   STAT0[201] := W#16#0;
   STAT0[202] := W#16#0;
   STAT0[203] := W#16#0;
   STAT0[204] := W#16#0;
   STAT0[205] := W#16#0;
   STAT0[206] := W#16#0;
   STAT0[207] := W#16#0;
   STAT0[208] := W#16#0;
   STAT0[209] := W#16#0;
   STAT0[210] := W#16#0;
   STAT0[211] := W#16#0;
   STAT0[212] := W#16#0;
   STAT0[213] := W#16#0;
   STAT0[214] := W#16#0;
   STAT0[215] := W#16#0;
   STAT0[216] := W#16#0;
   STAT0[217] := W#16#0;
   STAT0[218] := W#16#0;
   STAT0[219] := W#16#0;
   STAT0[220] := W#16#0;
   STAT0[221] := W#16#0;
   STAT0[222] := W#16#0;
   STAT0[223] := W#16#0;
   STAT0[224] := W#16#0;
   STAT0[225] := W#16#0;
   STAT0[226] := W#16#0;
   STAT0[227] := W#16#0;
   STAT0[228] := W#16#0;
   STAT0[229] := W#16#0;
   STAT0[230] := W#16#0;
   STAT0[231] := W#16#0;
   STAT0[232] := W#16#0;
   STAT0[233] := W#16#0;
   STAT0[234] := W#16#0;
   STAT0[235] := W#16#0;
   STAT0[236] := W#16#0;
   STAT0[237] := W#16#0;
   STAT0[238] := W#16#0;
   STAT0[239] := W#16#0;
   STAT0[240] := W#16#0;
   STAT0[241] := W#16#0;
   STAT0[242] := W#16#0;
   STAT0[243] := W#16#0;
   STAT0[244] := W#16#0;
   STAT0[245] := W#16#0;
   STAT0[246] := W#16#0;
   STAT0[247] := W#16#0;
   STAT0[248] := W#16#0;
   STAT0[249] := W#16#0;
   STAT0[250] := W#16#0;
   STAT0[251] := W#16#0;
   STAT0[252] := W#16#0;
   STAT0[253] := W#16#0;
   STAT0[254] := W#16#0;
   STAT0[255] := W#16#0;
END_DATA_BLOCK

DATA_BLOCK DB 51
TITLE =
VERSION : 0.1


